Universal Robots PolyScope program: Cube.urp

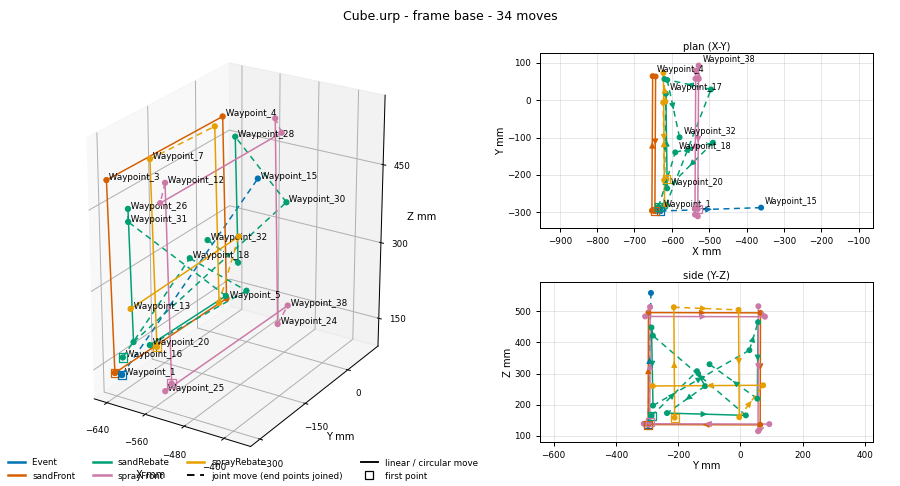
[picture p0: tool path of Cube.urp in frame base, 34 of 34 moves have a stored position in this frame; points joined in program order, loops and branches not executed]
Program Cube (installation=Cube directory=/programs/cube/archive createdIn=5.11.5.1010327 lastSavedIn=5.11.5.1010327 robotSerialNumber=20215500677)
Calibrated DH parameters: a=[0.000204, -0.239222, -0.391845, -0.000001, 0.000022, 0]; d=[0.162722, -355.808559, 353.37206, 2.570385, 0.099741, 0.099629]; alpha=[1.571124, 0.000988, 0.008295, 1.568963, -1.570303, 0]; deltaTheta=[0, -0.973091, 7.204745, 0.05153, 0, 0]
Robot Program (runOnlyOnce=false)
  Set DigitalOutput pin=digital_out[6]; digitalValue=1
  Wait Sleep waitTime=0.01
SuppressedNode
  SubProgram Sand45 (keepSynchronizedWithDisk=false)
    MoveJ speed 60 deg/s, acceleration 80 deg/s^2 (useActiveTCP=false) tcp=SandTCP; feature=Base
      Waypoint Waypoint_33: TCP in base x=552.09 y=70.738 z=404 mm, rx=2.2788 ry=-2.1615 rz=0.0012 rad; joints [23.825, -116.535, -41.178, 110.72, -75.887, -164.688] deg; TCP offset x=3.18 y=114.64 z=98.2 mm, rx=-0.7854 ry=0 rz=0 rad
      URCap Find Surface (Robotiq_Copilot, Robotiq Inc.) dataModel(NodeInitializedKey=true, WaitForSteadyWrenchOptionKey=false, ls_force=10.0, ls_distance=100.0, ls_speed=5.0, HackTriggeringContributionIsDefinedMethodKey=true, ZeroSensorBeforeKey=true, ls_if_distance=false, ls_if_force=false); state(isChildrenLocked=true)
        'Add Stop conditions from the Find Surface node'
      Force Simple feature=Joint_6_name; selection=[0, 0, 1, 0, 0, 0]; wrench=[0, 0, 1, 0, 0, 0]; limitsForce=[0.15, 0.15, 0.15, 1.047198, 1.047198, 1.047198]; limitsMotion=[0.1, 0.1, 0.1, 0.349066, 0.349066, 0.349066]
        MoveL speed 60 mm/s, acceleration 1200 mm/s^2 (useActiveTCP=false) tcp=SandTCP; feature=CubeFront
          Waypoint Waypoint_34: TCP in base x=-615.869 y=17.644 z=165.5 mm, rx=-0.1405 ry=3.133 rz=-0.0083 rad; joints [-19.498, -69.391, 89.408, 273.085, -49.409, -123.045] deg; feature pose in base x=-655.522 y=-293.872 z=132.154 mm, rx=1.1865 ry=1.2078 rz=1.229 rad
          URCap Finishing Tool Control (Robotiq_Copilot, Robotiq Inc.) dataModel(FinishingToolStateKey=false, ToolOutputNameKey=SanderOn, HackTriggeringContributionIsDefinedMethodKey=true)
Event  expression=digital_in[2]≟ True
  Set DigitalOutput pin=digital_out[7]; digitalValue=1
  MoveJ speed 60 deg/s, acceleration 80 deg/s^2 (useActiveTCP=false) tcp=SandTCP; feature=CubeFront
    Waypoint Waypoint_1: TCP in base x=-630.407 y=-296.529 z=136.222 mm, rx=-1.2299 ry=-1.2202 rz=1.1966 rad; joints [21.158, -27.557, 89.423, 72.355, -105.869, -15.062] deg; feature pose in base x=-655.41 y=-296.377 z=135.695 mm, rx=1.1937 ry=1.1902 rz=1.2137 rad
  Call sandFront
  Call sandFront
  SuppressedNode
    Call sandRebate
  SuppressedNode
    Call sandRebate
  MoveJ speed 60 deg/s, acceleration 80 deg/s^2 (useActiveTCP=false) tcp=SandTCP; feature=CubeFront
    Waypoint Waypoint_1: TCP in base x=-630.407 y=-296.529 z=136.222 mm, rx=-1.2299 ry=-1.2202 rz=1.1966 rad; joints [21.158, -27.557, 89.423, 72.355, -105.869, -15.062] deg
  Call sprayFront
  Call sprayRebate
  Set DigitalOutput pin=digital_out[7]; digitalValue=0
  MoveJ speed 60 deg/s, acceleration 80 deg/s^2 (useActiveTCP=false) tcp=SprayTCP; feature=Base
    Waypoint Waypoint_15: TCP in base x=-361.118 y=-287.404 z=558.951 mm, rx=1.2298 ry=-1.2143 rz=-1.1943 rad; joints [31.296, -74.431, 112.566, 95.409, -108.908, -17.973] deg; TCP offset x=20.839 y=-27.14 z=105.994 mm, rx=0.1226 ry=1.1769 rz=2.8697 rad
SubProgram -> sandRebate
SubProgram -> sprayRebate
SubProgram -> sprayFront
SubProgram -> sandFront
SubProgram sandFront (keepSynchronizedWithDisk=true) programFile=/programs/April2022Sand/subs/sandFront.urp
  Folder sandFront
    Set NoAction tcp=SandTCP
    MoveL speed 250 mm/s, acceleration 1200 mm/s^2 (useActiveTCP=false) tcp=SandTCP; feature=CubeFront
      Waypoint Waypoint_2: TCP in base x=-645.398 y=-296.455 z=135.894 mm, rx=-1.2299 ry=-1.2203 rz=1.1965 rad; joints [20.532, -26.698, 86.988, 74.06, -105.434, -14.586] deg; TCP offset x=3.18 y=114.64 z=98.2 mm, rx=-0.7854 ry=0 rz=0 rad; feature pose in base x=-150.564 y=-110.257 z=792.369 mm, rx=-0.0207 ry=-0.0133 rz=3.0697 rad
      URCap Zero FT Sensor (Robotiq_Copilot, Robotiq Inc.) dataModel(NodeInitializedKey=true, WaitForSteadyWrenchOptionKey=true, HackTriggeringContributionIsDefinedMethodKey=true)
      MoveDirectionNode (selectedDirection=ZPlus toolParams=0.05, 1.2) feature=Joint_6_name
        Until TOOL_CONTACT_DETECTION (allowActions=false retraction=NONE decelerationAcceleration=3 decelerationAngularAcceleration=34.906585)
      URCap Finishing Tool Control (Robotiq_Copilot, Robotiq Inc.) dataModel(ToolOutputNameKey=SanderOn, HackTriggeringContributionIsDefinedMethodKey=true)
      Wait Sleep waitTime=1
    MoveL speed 120 mm/s, acceleration 1200 mm/s^2 (useActiveTCP=false) tcp=SandTCP; feature=CubeFront
      URCap Zero FT Sensor (Robotiq_Copilot, Robotiq Inc.) dataModel(NodeInitializedKey=true, WaitForSteadyWrenchOptionKey=false, HackTriggeringContributionIsDefinedMethodKey=true)
      Force Simple feature=Joint_6_name; selection=[0, 0, 1, 0, 0, 0]; wrench=[0, 0, 1, 0, 0, 0]; limitsForce=[0.15, 0.15, 0.15, 1.047198, 1.047198, 1.047198]; limitsMotion=[0.1, 0.1, 0.1, 0.349066, 0.349066, 0.349066]
        Waypoint Waypoint_3: TCP in base x=-653.335 y=-295.509 z=495.795 mm, rx=-1.2297 ry=-1.2204 rz=1.1965 rad; joints [20.051, -59.037, 82.186, 111.364, -105.042, -13.942] deg
        Waypoint Waypoint_4: TCP in base x=-651.379 y=64.515 z=494.966 mm, rx=-1.2297 ry=-1.2202 rz=1.1965 rad; joints [-25.966, -70.491, 99.418, 104.332, -72.274, 18.732] deg
        Waypoint Waypoint_5: TCP in base x=-643.444 y=63.548 z=135.045 mm, rx=-1.2296 ry=-1.2202 rz=1.1965 rad; joints [-26.244, -31.945, 104.603, 60.633, -72.073, 18.608] deg
        Waypoint Waypoint_6: TCP in base x=-645.385 y=-296.43 z=135.968 mm, rx=-1.2296 ry=-1.2201 rz=1.1966 rad; joints [20.529, -26.7, 86.987, 74.045, -105.424, -14.592] deg
        URCap Finishing Tool Control (Robotiq_Copilot, Robotiq Inc.) dataModel(ToolOutputNameKey=SanderOn, FinishingToolStateKey=false, HackTriggeringContributionIsDefinedMethodKey=true)
      MoveDirectionNode (selectedDirection=ZMinus) feature=Joint_6_name
        Until DISTANCE (allowActions=false deceleration=3 distanceNodeType=STOP) Distance=0.025; motionParameters(blendRadius=0)
SubProgram sandRebate (keepSynchronizedWithDisk=false)
  MoveJ speed 60 deg/s, acceleration 80 deg/s^2 (useActiveTCP=false) tcp=SandTCP; feature=CubeFront
    Waypoint Waypoint_16: TCP in base x=-635.651 y=-285.476 z=163.792 mm, rx=-1.2268 ry=-1.2306 rz=1.2152 rad; joints [19.32, -31.087, 91.666, 74.12, -104.14, -12.636] deg; feature pose in base x=-660.434 y=-291.842 z=157.322 mm, rx=1.1794 ry=1.2066 rz=1.222 rad
    Waypoint Waypoint_18: TCP in base x=-590.751 y=-139.462 z=307.521 mm, rx=-1.2266 ry=-1.2307 rz=1.2152 rad; joints [1.031, -56.343, 114.796, 77.853, -91.029, 0.265] deg
    Waypoint Waypoint_19: TCP in base x=-489.992 y=-113.645 z=259.46 mm, rx=1.2012 ry=2.9028 rz=0.0002 rad; joints [-7.833, -91.59, 115.365, 214.849, -55.403, -42.538] deg
    Waypoint Waypoint_20: TCP in base x=-612.491 y=-235.853 z=172.874 mm, rx=-0.1406 ry=3.1331 rz=-0.0084 rad; joints [3.875, -66.825, 90.341, 247.878, -44.265, -91.522] deg; TCP offset x=3.18 y=114.64 z=98.2 mm, rx=-0.7854 ry=0 rz=0 rad
    URCap Find Surface (Robotiq_Copilot, Robotiq Inc.) dataModel(NodeInitializedKey=true, WaitForSteadyWrenchOptionKey=false, ls_force=10.0, ls_distance=100.0, ls_speed=5.0, HackTriggeringContributionIsDefinedMethodKey=true, ls_if_distance=false, ls_if_force=false, ZeroSensorBeforeKey=true); state(isChildrenLocked=true)
      'Add Stop conditions from the Find Surface node'
    URCap Finishing Tool Control (Robotiq_Copilot, Robotiq Inc.) dataModel(ToolOutputNameKey=SanderOn, HackTriggeringContributionIsDefinedMethodKey=true)
    Force Simple feature=Joint_6_name; selection=[0, 0, 1, 0, 0, 0]; wrench=[0, 0, 1, 0, 0, 0]; limitsForce=[0.15, 0.15, 0.15, 1.047198, 1.047198, 1.047198]; limitsMotion=[0.1, 0.1, 0.1, 0.349066, 0.349066, 0.349066]
      MoveL speed 60 mm/s, acceleration 1200 mm/s^2 (useActiveTCP=false) tcp=SandTCP; feature=CubeFront
        Waypoint Waypoint_17: TCP in base x=-615.869 y=17.644 z=165.5 mm, rx=-0.1405 ry=3.133 rz=-0.0083 rad; joints [-19.498, -69.391, 89.408, 273.085, -49.409, -123.045] deg; TCP offset x=3.18 y=114.64 z=98.2 mm, rx=-0.7854 ry=0 rz=0 rad
        URCap Finishing Tool Control (Robotiq_Copilot, Robotiq Inc.) dataModel(FinishingToolStateKey=false, ToolOutputNameKey=SanderOn, HackTriggeringContributionIsDefinedMethodKey=true)
    MoveL speed 250 mm/s, acceleration 1200 mm/s^2 (useActiveTCP=true) feature=Base
      MoveDirectionNode (selectedDirection=ZMinus) feature=Joint_6_name
        Until DISTANCE (allowActions=false deceleration=3 distanceNodeType=STOP) Distance=0.1; motionParameters(blendRadius=0)
      MoveDirectionNode (selectedDirection=ZPlus) feature(featureName=CubeFront)
        Until DISTANCE (allowActions=false deceleration=3 distanceNodeType=STOP) Distance=0.15; motionParameters(blendRadius=0)
    MoveJ speed 60 deg/s, acceleration 80 deg/s^2 (useActiveTCP=false) tcp=SandTCP; feature=CubeFront
      Waypoint Waypoint_31: TCP in base x=-620.705 y=-281.439 z=421.856 mm, rx=0.4422 ry=-1.9578 rz=1.8694 rad; joints [-6.993, -60.978, 93.613, 204.92, 45.478, -85.559] deg
      Waypoint Waypoint_26: TCP in base x=-617.598 y=-285.662 z=447.888 mm, rx=0.2579 ry=-2.0809 rz=2.0837 rad; joints [-6.389, -64.912, 93.992, 221.227, 47.236, -82.684] deg; feature pose in base x=-655.41 y=-296.377 z=135.695 mm, rx=1.1937 ry=1.1902 rz=1.2137 rad
    URCap Find Surface (Robotiq_Copilot, Robotiq Inc.) dataModel(NodeInitializedKey=true, WaitForSteadyWrenchOptionKey=false, ls_force=10.0, ls_distance=100.0, ls_speed=5.0, ZeroSensorBeforeKey=true, ls_if_distance=false, ls_if_force=false, HackTriggeringContributionIsDefinedMethodKey=true); state(isChildrenLocked=true)
      'Add Stop conditions from the Find Surface node'
    URCap Finishing Tool Control (Robotiq_Copilot, Robotiq Inc.) dataModel(ToolOutputNameKey=SanderOn, HackTriggeringContributionIsDefinedMethodKey=true)
    Force Simple feature=Joint_6_name; selection=[0, 0, 1, 0, 0, 0]; wrench=[0, 0, 1, 0, 0, 0]; limitsForce=[0.15, 0.15, 0.15, 1.047198, 1.047198, 1.047198]; limitsMotion=[0.1, 0.1, 0.1, 0.349066, 0.349066, 0.349066]
      MoveL speed 60 mm/s, acceleration 1200 mm/s^2 (useActiveTCP=false) tcp=SandTCP; feature=CubeFront
        Waypoint Waypoint_27: TCP in base x=-615.451 y=-280.884 z=196.979 mm, rx=0.1862 ry=2.2283 rz=-2.172 rad; joints [-7.314, -49.403, 108.062, 213.951, 43.385, -85.69] deg; TCP offset x=3.18 y=114.64 z=98.2 mm, rx=-0.7854 ry=0 rz=0 rad; feature pose in base x=-660.434 y=-291.842 z=157.322 mm, rx=1.1794 ry=1.2066 rz=1.222 rad
        URCap Finishing Tool Control (Robotiq_Copilot, Robotiq Inc.) dataModel(FinishingToolStateKey=false, ToolOutputNameKey=SanderOn, HackTriggeringContributionIsDefinedMethodKey=true)
    MoveL speed 250 mm/s, acceleration 1200 mm/s^2 (useActiveTCP=true) feature=Base
      MoveDirectionNode (selectedDirection=ZMinus) feature=Joint_6_name
        Until DISTANCE (allowActions=false deceleration=3 distanceNodeType=STOP) Distance=0.05; motionParameters(blendRadius=0)
      MoveDirectionNode (selectedDirection=ZPlus) feature(featureName=CubeFront)
        Until DISTANCE (allowActions=false deceleration=3 distanceNodeType=STOP) Distance=0.15; motionParameters(blendRadius=0)
    MoveJ speed 60 deg/s, acceleration 80 deg/s^2 (useActiveTCP=false) tcp=SandTCP; feature=CubeFront
      Waypoint Waypoint_30: TCP in base x=-495.207 y=28.979 z=374.875 mm, rx=-1.178 ry=-1.4293 rz=-1.1379 rad; joints [6.71, -80.185, 91.347, 2.423, 134.71, 101.731] deg; TCP offset x=3.18 y=114.64 z=98.2 mm, rx=-0.7854 ry=0 rz=0 rad
      Waypoint Waypoint_28: TCP in base x=-619.839 y=56.782 z=465.017 mm, rx=-1.0386 ry=-1.45 rz=-1.4226 rad; joints [3.083, -60.105, 53.348, 26.397, 136.774, 92.25] deg; TCP offset x=3.18 y=114.64 z=98.2 mm, rx=-0.7854 ry=0 rz=0 rad
    URCap Find Surface (Robotiq_Copilot, Robotiq Inc.) dataModel(NodeInitializedKey=true, WaitForSteadyWrenchOptionKey=false, ls_force=10.0, ls_distance=100.0, ls_speed=5.0, ZeroSensorBeforeKey=true, ls_if_distance=false, ls_if_force=false, HackTriggeringContributionIsDefinedMethodKey=true); state(isChildrenLocked=true)
      'Add Stop conditions from the Find Surface node'
    URCap Finishing Tool Control (Robotiq_Copilot, Robotiq Inc.) dataModel(ToolOutputNameKey=SanderOn, HackTriggeringContributionIsDefinedMethodKey=true)
    Force Simple feature=Joint_6_name; selection=[0, 0, 1, 0, 0, 0]; wrench=[0, 0, 1, 0, 0, 0]; limitsForce=[0.15, 0.15, 0.15, 1.047198, 1.047198, 1.047198]; limitsMotion=[0.1, 0.1, 0.1, 0.349066, 0.349066, 0.349066]
      MoveL speed 100 mm/s, acceleration 1200 mm/s^2 (useActiveTCP=false) tcp=SandTCP; feature=CubeFront
        Waypoint Waypoint_29: TCP in base x=-612.287 y=54.274 z=219.23 mm, rx=-1.5598 ry=-0.2733 rz=-0.2501 rad; joints [3.146, -52.244, 103.361, -124.549, 136.519, 86.512] deg; TCP offset x=3.18 y=114.64 z=98.2 mm, rx=-0.7854 ry=0 rz=0 rad
        URCap Finishing Tool Control (Robotiq_Copilot, Robotiq Inc.) dataModel(FinishingToolStateKey=false, ToolOutputNameKey=SanderOn, HackTriggeringContributionIsDefinedMethodKey=true)
    MoveL speed 250 mm/s, acceleration 1200 mm/s^2 (useActiveTCP=true) feature=Base
      MoveDirectionNode (selectedDirection=ZMinus) feature=Joint_6_name
        Until DISTANCE (allowActions=false deceleration=3 distanceNodeType=STOP) Distance=0.05; motionParameters(blendRadius=0)
      MoveDirectionNode (selectedDirection=ZPlus) feature(featureName=CubeFront)
        Until DISTANCE (allowActions=false deceleration=3 distanceNodeType=STOP) Distance=0.15; motionParameters(blendRadius=0)
    MoveJ speed 60 deg/s, acceleration 80 deg/s^2 (useActiveTCP=true) feature=Base
      Waypoint Waypoint_32: TCP in base x=-579.374 y=-99.248 z=329.851 mm, rx=-1.0804 ry=-1.2563 rz=0.9494 rad; joints [-3.921, -93.741, 131.693, -81.717, 81.638, 168.644] deg; TCP offset x=3.18 y=114.64 z=98.2 mm, rx=-0.7854 ry=0 rz=0 rad
SubProgram sprayFront (keepSynchronizedWithDisk=true) programFile=/programs/April2022Sand/subs/sprayFront.urp
  Folder SprayFront
    MoveJ speed 60 deg/s, acceleration 80 deg/s^2 (useActiveTCP=false) tcp=SprayTCP; feature=CubeFront
      Waypoint Waypoint_10: TCP in base x=-530.531 y=-291.052 z=144.441 mm, rx=-2.2301 ry=-0.0105 rz=2.1935 rad; joints [-0.761, -65.891, 118.661, -46.487, 45.268, 89.493] deg; TCP offset x=20.839 y=-27.14 z=105.994 mm, rx=0.1226 ry=1.1769 rz=2.8697 rad; feature pose in base x=-150.564 y=-110.257 z=792.369 mm, rx=-0.0207 ry=-0.0133 rz=3.0697 rad
      Set DigitalOutput pin=SprayerOn; digitalValue=1
    MoveL speed 100 mm/s, acceleration 1200 mm/s^2 (useActiveTCP=true) feature=CubeFront
      Waypoint Waypoint_12: TCP in base x=-538.683 y=-290.104 z=513.862 mm, rx=-2.2302 ry=-0.0105 rz=2.1934 rad; joints [-0.84, -86.478, 83.393, 9.273, 44.774, 89.634] deg
      Set DigitalOutput pin=SprayerOn; digitalValue=0
      MoveDirectionNode (selectedDirection=ZMinus toolParams=0.2, 1.2) feature=Joint_6_name
        Until DISTANCE (allowActions=false deceleration=3 distanceNodeType=STOP) Distance=0.1; motionParameters(blendRadius=0)
    MoveJ speed 60 deg/s, acceleration 80 deg/s^2 (useActiveTCP=false) tcp=SprayTCP; feature=CubeFront
      Waypoint Waypoint_21: TCP in base x=-538.097 y=-306.157 z=483.391 mm, rx=1.2299 ry=-1.2185 rz=-1.2154 rad; joints [22.708, -78.928, 107.314, -73.338, 103.019, 167.126] deg; TCP offset x=20.839 y=-27.14 z=105.994 mm, rx=0.1226 ry=1.1769 rz=2.8697 rad
      Set DigitalOutput pin=SprayerOn; digitalValue=1
    MoveL speed 100 mm/s, acceleration 1200 mm/s^2 (useActiveTCP=false) tcp=SprayTCP; feature=CubeFront
      Waypoint Waypoint_22: TCP in base x=-536.01 y=78.845 z=482.449 mm, rx=1.2299 ry=-1.2184 rz=-1.2154 rad; joints [-28.836, -93.233, 123.857, -79.597, 66.516, 204.312] deg; TCP offset x=20.839 y=-27.14 z=105.994 mm, rx=0.1226 ry=1.1769 rz=2.8697 rad
      Set DigitalOutput pin=SprayerOn; digitalValue=0
      MoveDirectionNode (selectedDirection=ZMinus toolParams=0.2, 1.2) feature=Joint_6_name
        Until DISTANCE (allowActions=false deceleration=3 distanceNodeType=STOP) Distance=0.1; motionParameters(blendRadius=0)
    MoveJ speed 60 deg/s, acceleration 80 deg/s^2 (useActiveTCP=false) tcp=SprayTCP; feature=CubeFront
      Waypoint Waypoint_23: TCP in base x=-536.857 y=57.735 z=516.338 mm, rx=0.0075 ry=-1.5876 rz=-0.0151 rad; joints [-3.715, -89.488, 83.743, 1.67, 131.045, 270.018] deg; TCP offset x=20.839 y=-27.14 z=105.994 mm, rx=0.1226 ry=1.1769 rz=2.8697 rad
      Set DigitalOutput pin=SprayerOn; digitalValue=1
    MoveL speed 100 mm/s, acceleration 1200 mm/s^2 (useActiveTCP=false) tcp=SprayTCP; feature=CubeFront
      Waypoint Waypoint_24: TCP in base x=-528.032 y=56.71 z=114.659 mm, rx=0.0075 ry=-1.5874 rz=-0.0151 rad; joints [-3.717, -66.449, 123.019, -60.833, 131.469, 269.749] deg; TCP offset x=20.839 y=-27.14 z=105.994 mm, rx=0.1226 ry=1.1769 rz=2.8697 rad
      Set DigitalOutput pin=SprayerOn; digitalValue=0
      MoveDirectionNode (selectedDirection=ZMinus toolParams=0.2, 1.2) feature=Joint_6_name
        Until DISTANCE (allowActions=false deceleration=3 distanceNodeType=STOP) Distance=0.1; motionParameters(blendRadius=0)
    MoveJ speed 60 deg/s, acceleration 80 deg/s^2 (useActiveTCP=false) tcp=SprayTCP; feature=CubeFront
      Waypoint Waypoint_38: TCP in base x=-528.302 y=92.929 z=137.544 mm, rx=1.2295 ry=-1.2182 rz=-1.2157 rad; joints [-31.314, -39.364, 132.373, -142.669, 64.779, 205.918] deg
      Set DigitalOutput pin=SprayerOn; digitalValue=1
    MoveL speed 100 mm/s, acceleration 1200 mm/s^2 (useActiveTCP=false) tcp=SprayTCP; feature=CubeFront
      Waypoint Waypoint_25: TCP in base x=-530.503 y=-310.8 z=138.54 mm, rx=1.2295 ry=-1.2182 rz=-1.2157 rad; joints [23.481, -38.767, 115.153, -121.572, 103.542, 166.189] deg
      Set DigitalOutput pin=SprayerOn; digitalValue=0
      MoveDirectionNode (selectedDirection=ZMinus toolParams=0.2, 1.2) feature=Joint_6_name
        Until DISTANCE (allowActions=false deceleration=3 distanceNodeType=STOP) Distance=0.1; motionParameters(blendRadius=0)
SubProgram sprayRebate (keepSynchronizedWithDisk=true) programFile=/programs/April2022Sand/subs/sprayRebate.urp
  Folder SprayRebate
    MoveJ speed 60 deg/s, acceleration 80 deg/s^2 (useActiveTCP=false) tcp=SprayTCP; feature=CubeFront
      Waypoint Waypoint_14: TCP in base x=-614.395 y=-211.304 z=158.056 mm, rx=0.8919 ry=-1.3989 rz=0.8972 rad; joints [3.832, -69.113, 116.159, -49.553, 73.09, -85.388] deg
      Set DigitalOutput pin=SprayerOn; digitalValue=1
    MoveL speed 100 mm/s, acceleration 1200 mm/s^2 (useActiveTCP=true) feature=CubeFront
      Waypoint Waypoint_7: TCP in base x=-620.397 y=-213.913 z=513.046 mm, rx=0.892 ry=-1.3988 rz=0.8971 rad; joints [4.169, -85.315, 79.236, 3.53, 73.033, -85.264] deg
      Set DigitalOutput pin=SprayerOn; digitalValue=0
      MoveDirectionNode (selectedDirection=ZPlus toolParams=0.2, 1.2)
        Until DISTANCE (allowActions=false deceleration=3 distanceNodeType=STOP) Distance=0.1; motionParameters(blendRadius=0)
    MoveJ speed 60 deg/s, acceleration 80 deg/s^2 (useActiveTCP=false) tcp=SprayTCP; feature=CubeFront
      Waypoint Waypoint_8: TCP in base x=-623.058 y=-6.085 z=504.453 mm, rx=-1.5379 ry=0.9456 rz=1.5188 rad; joints [-11.433, -87.799, 86.311, 5.702, 98.013, 93.92] deg
      Set DigitalOutput pin=SprayerOn; digitalValue=1
    MoveL speed 100 mm/s, acceleration 1200 mm/s^2 (useActiveTCP=false) tcp=SprayTCP; feature=CubeFront
      Waypoint Waypoint_9: TCP in base x=-617.186 y=-3.636 z=159.537 mm, rx=-1.538 ry=0.9455 rz=1.5188 rad; joints [-11.994, -68.384, 119.511, -46.936, 97.835, 93.758] deg
      Set DigitalOutput pin=SprayerOn; digitalValue=0
      MoveDirectionNode (selectedDirection=ZPlus toolParams=0.2, 1.2)
        Until DISTANCE (allowActions=false deceleration=3 distanceNodeType=STOP) Distance=0.1; motionParameters(blendRadius=0)
    MoveJ speed 60 deg/s, acceleration 80 deg/s^2 (useActiveTCP=false) tcp=SprayTCP; feature=CubeFront
      Waypoint Waypoint_11: TCP in base x=-622.643 y=73.149 z=262.251 mm, rx=2.0067 ry=-1.985 rz=-0.4223 rad; joints [-27.089, -68.36, 126.552, 146.432, -61.498, -7.368] deg; TCP offset x=20.839 y=-27.14 z=105.994 mm, rx=0.1226 ry=1.1769 rz=2.8697 rad
      Set DigitalOutput pin=SprayerOn; digitalValue=1
    MoveL speed 100 mm/s, acceleration 1200 mm/s^2 (useActiveTCP=false) tcp=SprayTCP; feature=CubeFront
      Waypoint Waypoint_13: TCP in base x=-619.354 y=-281.828 z=259.921 mm, rx=2.0066 ry=-1.9851 rz=-0.4224 rad; joints [19.517, -59.938, 112.11, 150.357, -104.552, 371.006] deg; TCP offset x=20.839 y=-27.14 z=105.994 mm, rx=0.1226 ry=1.1769 rz=2.8697 rad
      Set DigitalOutput pin=SprayerOn; digitalValue=0
      MoveDirectionNode (selectedDirection=ZPlus toolParams=0.2, 1.2)
        Until DISTANCE (allowActions=false deceleration=3 distanceNodeType=STOP) Distance=0.1; motionParameters(blendRadius=0)
